(* Logix 5000 project; controller Planta_de_Kumis vendor 1 type 14 code 54 rev 20.11; software revision 20.00 *)

TASK Mapeo_IO (periodic, rate 10 ms, priority 6, watchdog 500 ms) : Mapeo_CadSim_Plus
TASK Rutina (periodic, rate 50 ms, priority 8, watchdog 500 ms) : MainProgram

MODULES
   Local : vendor 1 type 14 code 54 (ICP 0, rev 20.11)
END_MODULES

VAR_GLOBAL   (* controller tags *)
   Azucar : BOOL;
   Cultivo : BOOL;
   CV_TCV_201_1 : REAL;
   CV_TCV_202_1 : REAL;
   FI_01 : REAL;   // Indicador de flujo del vapor Intercambiador 1
   FI_02 : REAL;   // Indicador de flujo del agua Intercambiador 2
   FT_1 : REAL;
   HV2 : REAL;   // Valvula de desfogue
   HV3 : REAL;   // Valvula de desfogue TK2
   HV4 : REAL;   // Valvula de desfogue TK3
   HV5 : REAL;   // Valvula de desfogue TK4
   HV6 : REAL;   // Valvula de desfogue TK5
   HV7 : REAL;   // Valvula de desfogue TK6
   HV8 : REAL;   // Valvula de desfogue TK7
   HV9 : REAL;   // Valvula de desfogue TK8
   JY_01 : BOOL;   // Motor de mezclado M1
   JY_02 : BOOL;   // Motor de mezclado cultivo
   KP_A : REAL;   // KP de letapa de aumento de temperatura
   KP_D : REAL;   // KP de etapa de disminucion de temperatura
   Leve_TK1 : REAL;   // Sensor de nivel TK1
   Level_TK10 : REAL;   // Sensor de nivel TK10 Intercambiador 2
   Level_TK2 : REAL;   // Sensor de nivel TK2
   Level_TK3 : REAL;   // Sensor de nivel TK·
   Level_TK4 : REAL;   // Sensor de nivel TK4
   Level_TK5 : REAL;   // Sensor de nivel TK5
   Level_TK6 : REAL;   // Sensor de nivel TK6
   Level_TK7 : REAL;   // Sensor de nivel TK7
   Level_TK8 : REAL;   // Sensor de nivel TK8
   Level_TK9 : REAL;   // Sensor de nivel TK9 Intercambiador 1
   LSH_101_1 : BOOL;   // Sensor de nivel alto TK1
   LSH_102_1 : BOOL;   // Sensor de nivel alto TK2
   LSH_103_1 : BOOL;   // Sensor de nivel alto TK3
   LSH_104_1 : BOOL;   // Sensor de nivel alto TK4
   LSH_105_1 : BOOL;   // Sensor de nivel alto TK5
   LSH_106_1 : BOOL;   // Sensor de nivel alto TK6
   LSH_107_1 : BOOL;   // Sensor de nivel alto TK7
   LSH_108_1 : BOOL;   // Sensor de nivel alto TK8
   LSL_101_1 : BOOL := 1;   // Sensor de nivel bajo TK1
   LSL_102_1 : BOOL := 1;   // Sensor de nivel bajo TK2
   LSL_103_1 : BOOL := 1;   // Sensor de nivel bajo TK3
   LSL_104_1 : BOOL := 1;   // Sensor de nivel bajo TK4
   LSL_105_1 : BOOL := 1;   // Sensor de nivel bajo TK5
   LSL_106_1 : BOOL := 1;   // Sensor de nivel bajo TK6
   LSL_107_1 : BOOL := 1;   // Sensor de nivel baj TK7
   LSL_108_1 : BOOL := 1;   // Sensor de nivel bajo TK8
   PI_01 : REAL;   // Indicador de presion del vapor Intercambiador 1
   PI_02 : REAL;   // Indicador de presion del agua Intercambiador 2
   PP1 : BOOL;   // Motobomba 1
   PP2 : BOOL;   // Motobomba 2
   PP3 : BOOL;   // Motobomba 3
   PP4 : BOOL;   // Motobomba 4
   PP5 : BOOL;   // Motobomba 5
   Reset : BOOL;
   SP_A : REAL;   // SETPOINT de letapa de aumento de temperatura
   SP_D : REAL;   // SETPOINT de etapa de disminucion de temperatura
   Start : BOOL;   // Boton de Inicio
   SV_101_1 : REAL;   // Valvula de salida TK1
   SV_102_1 : REAL;   // Valvula de salida TK2
   SV_103_1 : REAL;   // Valvula de salida TK3
   SV_104_1 : REAL;   // Valvula de salida
   SV_105_1 : REAL;   // Valvula de entrada TK5
   SV_106_1 : REAL;   // Valvula de entrada TK6
   SV_107_1 : REAL;   // Valvula de entrada TK7
   SV_108_1 : REAL;   // Valvula de entrada TK8
   SV_201_1 : REAL;   // Valvula de salida 1 Intercambiador
   SV_201_2 : REAL;   // Valvula de reflujo Intercambiador 1
   SV_202_1 : REAL;   // Valvula de salida 1 Intercambiador 2
   SV_202_2 : REAL;   // Valvula de reflujo
   T_Agua : DINT := 4;   // Temperatura de entrada del Agua Fria
   T_Int : DINT := 18;   // Temperatura de entrada de la leche
   TCV_101_1 : REAL;   // Valvula de entrada de Leche Variable manipulada
   TCV_201_1 : REAL;
   TCV_202_1 : REAL;   // Valvula de entrada de agua Variable manipulada Intercambiador 2
   TD_A : REAL;   // TD de letapa de aumento de temperatura
   TD_D : REAL;   // TD de etapa de disminucion de temperatura
   TI_01 : REAL;   // Indicador de temperatura TK1
   TI_02 : REAL;   // Indicador de temperatura TK2
   TI_03 : REAL;   // Indicador de temperatura del vapor Intercambiador 1
   TI_05 : REAL;   // Indicador de temperatura TK3
   TI_06 : REAL;   // Indicador de temperatura del agua
   TI_A : REAL;   // TI de letapa de aumento de temperatura
   TI_D : REAL;   // TI de etapa de disminucion de temperatura
   TITE_201_1 : REAL;   // Sensor de temperatura de producto intermedio Variable Controlada Intercambiador 1
   TITE_202_1 : REAL;   // Sensor de temperatura de producto intermedio Variable controlada Intercambiador 2
   TITE_Prueba : REAL;
   TITE_Prueba_2 : REAL;
END_VAR

PROGRAM MainProgram   (* main routine MainRoutine *)
VAR
   a1_A : REAL;   // parametro del modelo del proceso discreto
   a1_D : REAL;   // Parametro del modelo del proceso discreto etapa de disminucion de temperatura
   aF1_A : REAL;   // Parametro delnumerador del filtro 1
   aF2_A : REAL;   // Parametro del filtro1
   b0_A : REAL;   // parametro del modelo del proceso discreto
   b0_D : REAL;   // Parametro del modelo del proceso discreto etapa de disminucion de temperatura
   b1_A : REAL;   // Parametros del modelo discreto del proceso
   b1_D : REAL;   // Parametro del modelo del proceso discreto etapa de disminucion de temperatura
   bF0_A : REAL;   // Parametro del filtro 1
   bF1_A : REAL;   // Parametro del filtro 1
   bF2_A : REAL;   // Parametro del filtro 1
   BIT_ACT : BOOL;   // BIT DE ACTIVACION ETAPA 0
   BIT_ACT2 : BOOL;   // BIT DE ACTIVACION ETAPA 0 Disminucion de temperatura
   BIT_MEZC_AZUCAR : BOOL;   // Indicador de mezclado de azucar
   BIT_MEZC_CULTIVO : BOOL;   // Bit indicador mezclado de cultivo
   BIT_PRUEBA : BOOL;
   BIT_PRUEBA_2 : BOOL;
   C1 : COUNTER := (PRE := 5);
   da : DINT;   // Retardo discreo etapa de aumento de temperatura
   dd : DINT;   // Retardo discreo etapa de disminucion de temperatura
   E0_A : REAL;   // Error actual en etapa de aumento de temperatura
   E0_D : REAL;   // Error actual en etapa de disminucion de temperatura
   E1_A : REAL;   // Error 1 instante pasado etapa de aumento de temperatura
   E1_D : REAL;   // Error 1 instante pasado etapa de disminucion de temperatura
   E2_A : REAL;   // Error 2 instantes pasados etapa de aumento de temperatura
   E2_D : REAL;   // Error 2 instantes pasados etapa de disminucion de temperatura
   Ep1_A : REAL;   // Error de prediccion 1 instante antes
   Ep2_A : REAL;   // Error de prediccion 2 instantes antes
   Ep_A : REAL;   // Error de prediccion etapa de aumento de temperatura
   Ep_D : REAL;   // Error de prediccion etapa de disminucion de temperatura
   ETAPA0_A : BOOL;   // Etapa 0 en etapa de aumento de temperatura
   ETAPA0_D : BOOL;   // Etapa 0 en etapa de disminucion de temperatura
   ETAPA10_A : BOOL;   // Etapa 10 de etapa de aumento de temperatura
   ETAPA10_D : BOOL;   // Etapa 10 en etapa de disminucion de temperatura
   ETAPA11_A : BOOL;   // Etapa 11 de etapa de aumento de temperatura
   ETAPA11_D : BOOL;   // Etapa 11 en etapa de disminucion de temperatura
   ETAPA12_A : BOOL;   // Etapa 12 de etapa de aumento de temperatura
   ETAPA12_D : BOOL;   // Etapa 12 en etapa de disminucion de temperatura
   ETAPA13_A : BOOL;   // Etapa 13 de etapa de aumento de temperatura
   ETAPA13_D : BOOL;   // Etapa 13 en etapa de disminucion de temperatura
   ETAPA14_A : BOOL;   // Etapa 14 en etapa de aumento de temperatura
   ETAPA14_D : BOOL;   // Etapa 14 en etapa de disminucion de temperatura
   ETAPA1_A : BOOL;   // Etapa 1 en etapa de aumento de temperatura
   ETAPA1_D : BOOL;   // Etapa 1 en etapa de disminucion de temperatura
   ETAPA2_A : BOOL;   // Etapa 2 en etapa de aumento de temperaura
   ETAPA2_D : BOOL;   // Etapa 2 en etapa de disminucion de temperatura
   ETAPA3_A : BOOL;   // Etapa 3 en etapa de aumento de temperatura
   ETAPA3_D : BOOL;   // Etapa 3 en etapa de disminucion de temperatura
   ETAPA4_A : BOOL;   // Etapa 4 en etapa de aumento de temperatura
   ETAPA4_D : BOOL;   // Etapa 4 en etapa de disminucion de temperatura
   ETAPA5_A : BOOL;   // Etapa 5 de etapa de aumento de temperatura
   ETAPA5_D : BOOL;   // Etapa 5 en etapa de disminucion de temperatura
   ETAPA6_A : BOOL;   // Etapa 6 de etapa de aumento de temperatura
   ETAPA6_D : BOOL;   // Etapa 6 en etapa de disminucion de temperatura
   ETAPA7_A : BOOL;   // Etapa 7 en etapa de aumento de temperatura
   ETAPA7_D : BOOL;   // Etapa 7 en etapa de disminucion de temperatura
   ETAPA8_A : BOOL;   // Etapa 8 en etapa de aumento de temperatura
   ETAPA8_D : BOOL;   // Etapa 8 en etapa de disminucion de temperatura
   ETAPA9_A : BOOL;   // Etapa 9 de etapa de aumento de temperatura
   ETAPA9_D : BOOL;   // Etapa 9 en etapa de disminucion de temperatura
   I_A : DINT;   // Indice etapa de aumento de temperatura
   I_D : DINT;   // Indice etapa de disminucion de temperatura
   KTA : DINT;   // Tiempo discreto actual ultima posicion del vector U etapa de aumento
   KTD : DINT;   // Tiempo discreto actual ultima posicion del vector U etapa de disminucion de temperatura
   Latch_Azcuar_On : BOOL;
   Latch_LSH_TK1 : BOOL;
   Latch_LSH_TK2 : BOOL;
   Latch_LSH_TK3 : BOOL;
   Latch_LSH_TK4 : BOOL;
   Latch_LSH_TK5 : BOOL;
   Latch_LSH_TK6 : BOOL;
   Latch_LSH_TK7 : BOOL;
   Latch_LSH_TK8 : BOOL;
   Latch_OSR_2 : BOOL;
   Latch_OSR_4 : BOOL;
   Latch_OSR_6 : BOOL;
   Latch_OSR_8 : BOOL;
   Latch_PID2 : BOOL;
   Latch_SR1 : BOOL;
   Latch_SR2 : BOOL;
   Latch_Timer_Mezclado_DN : BOOL;
   Next_Batch : BOOL;
   OSR_1 : BOOL;
   OSR_2 : BOOL;
   OSR_3 : BOOL;
   OSR_4 : BOOL;
   OSR_5 : BOOL;
   OSR_6 : BOOL;
   OSR_7 : BOOL;
   OSR_8 : BOOL;
   OSRI_1 : FBD_ONESHOT;   // PULSO
   OSRI_2 : FBD_ONESHOT;   // Pulso
   PID_Exchanger_1 : PID := (CTL := 142607488, DOE := 1, PE := 1, DVNA := 1, PVHA := 1, SP := 60.0, MAXS := 100.0, MINS := 18.0, MAXO := 100.0, UPD := 1.0, MAXI := 100.0, MINI := 18.0, MAXCV := 100.0, DATA[0] := 45.327106, DATA[1] := -1256.7006, DATA[2] := 117.815674, DATA[3] := -57.815674, DATA[4] := 60.0, DATA[5] := 0.6666667, DATA[6] := 1.0, DATA[7] := 0.8, DATA[8] := 0.51, DATA[9] := 0.018, DATA[11] := 0.51, DATA[12] := 0.018, DATA[15] := 1.5, DATA[16] := 0.024420025);   // PID para el intercambiado de calor con vapor
   PID_Exchanger_2 : PID := (CTL := 176165504, DOE := 1, CA := 1, PE := 1, OLH := 1, DVPA := 1, PVHA := 1, SP := 40.0, MAXS := 100.0, SO := 100.0, MAXO := 100.0, UPD := 1.0, ERR := 39.804905, MAXI := 100.0, MAXCV := 100.0, DATA[0] := 65.07602, DATA[1] := -0.31215367, DATA[2] := 0.19509344, DATA[3] := 39.804905, DATA[4] := 40.0, DATA[5] := 0.1, DATA[6] := 1.0, DATA[7] := 33.989998, DATA[8] := 0.013, DATA[9] := 71.98, DATA[10] := 17.99, DATA[11] := 0.013, DATA[12] := 71.98, DATA[13] := 17.99, DATA[15] := 10.0, DATA[16] := 0.024420025);   // PID para el intercambiador de disminucion de temperatura
   q0_A : REAL;   // Parametro del controlador PID digital
   q0_D : REAL;   // Parametro del controlador PID digital etapa de disminucion de temperatura
   q1_A : REAL;   // Parametros del controlador PID digital
   q1_D : REAL;   // Parametro del controlador PID digital etapa de disminucion de temperatura
   q2_A : REAL;   // Parametros del controlador PID digital
   q2_D : REAL;   // Parametro del controlador PID digital etapa de disminucion de temperatura
   Salida_Prueba_1 : BOOL;
   TIMER_AT : FBD_TIMER;   // Timer de espera para mover datos en el vector de esfuerzo de control etapa de aumento de temperatura
   Timer_Azucar : TIMER := (PRE := 1000);
   Timer_Cultivo : TIMER := (PRE := 1000);
   Timer_Disminucion_T : TIMER := (PRE := 1000);
   TIMER_DT : FBD_TIMER;   // Timer de espera para mover datos en el vector de esfuerzo de control etapa de disminucion de temperatura
   timer_Elevado_T : TIMER := (PRE := 1000);
   Timer_Inoculado : TIMER := (PRE := 6000);
   Timer_Latch_PID2 : TIMER := (PRE := 42000);   // Timer para activacion del PID 2
   Timer_Mezclado : TIMER := (PRE := 1000);
   Timer_Recepcion : TIMER := (PRE := 1000);
   Timer_TK5 : TIMER := (PRE := 5000);
   Timer_TK6 : TIMER := (PRE := 5000);
   Timer_TK7 : TIMER := (PRE := 5000);
   Timer_TK8 : TIMER := (PRE := 5000);
   Tm_A : REAL;   // Tiempo de muestreo etapa aumento de temperatura
   Tm_D : REAL;   // Tiempo de muestreo etapa disminucion de temperatura
   VEC_U_A : REAL[24];   // VECTOR DE ESFUERZO DE CONTROL de etapa de aumento de temperatura
   VEC_U_D : REAL[24];   // VECTOR DE ESFUERZO DE CONTROL de etapa de disminucion de temperatura
   yF1_A : REAL;   // salida del filtro 1 instante antes
   yF2_A : REAL;   // salida del filtro 1 endos instantes antes
   yF_A : REAL;   // Salida del filtro 1
   Yn1_A : REAL;   // Salida del modelo nominal (Con retardo) 1 instante antes etapa de aumento de temparatura
   Yn1_D : REAL;   // Salida del modelo nominal (Con retardo) 1 instante antes etapa de disminucion de temperatura
   Yn_A : REAL;   // Salida del modelo nominal (Con retardo) etapa de aumento de temperatura
   Yn_D : REAL;   // Salida del modelo nominal (Con retardo) etapa de disminucion de temperatura
   Yp_A : REAL;   // Salida predicha etapa de aumento de temperatura
   Yp_D : REAL;   // Salida predicha etapa de disminucion de temperatura
   Yt1_A : REAL;   // Salida del modelo nominal rapido (Sin retardo) 1 instante antes etapa de aumento de temperatura
   Yt1_D : REAL;   // Salida del modelo nominal rapido (Sin retardo) 1 instante antes etapa de disminucion de temperatura
   Yt_A : REAL;   // Salida del modelo nominal rapido (Sin retardo) etapa de aumento de temperatura
   Yt_D : REAL;   // Salida del modelo nominal rapido (Sin retardo) etapa de disminucion de temperatura
END_VAR

ROUTINE MainRoutine   (* ladder *)
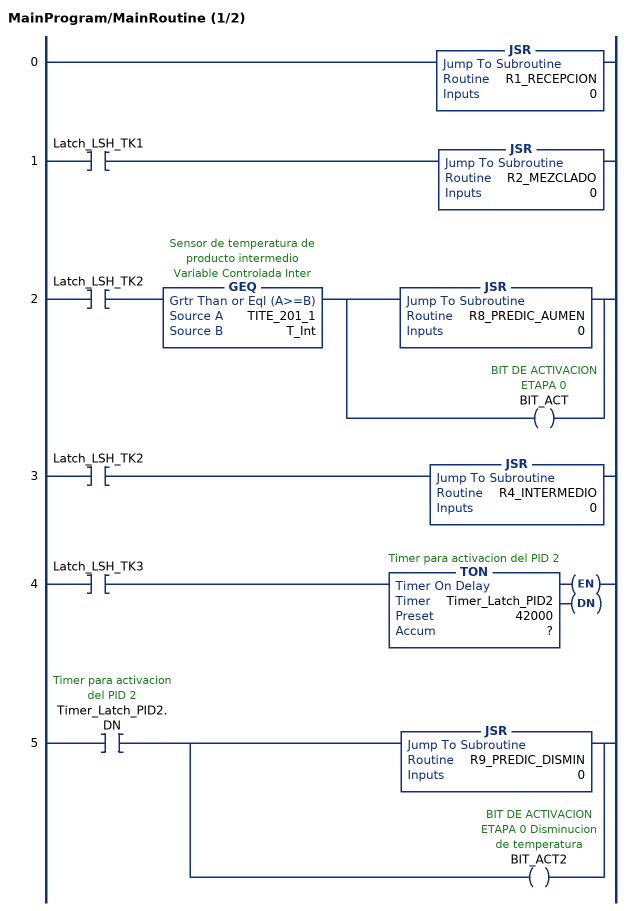
   0: JSR(R1_RECEPCION,0);
   1: XIC(Latch_LSH_TK1)JSR(R2_MEZCLADO,0);
   2: XIC(Latch_LSH_TK2)GEQ(TITE_201_1,T_Int)[JSR(R8_PREDIC_AUMEN,0) ,OTE(BIT_ACT) ];
   3: XIC(Latch_LSH_TK2)JSR(R4_INTERMEDIO,0);
   4: XIC(Latch_LSH_TK3)TON(Timer_Latch_PID2,?,?);
   5: XIC(Timer_Latch_PID2.DN)[JSR(R9_PREDIC_DISMIN,0) ,OTE(BIT_ACT2) ];
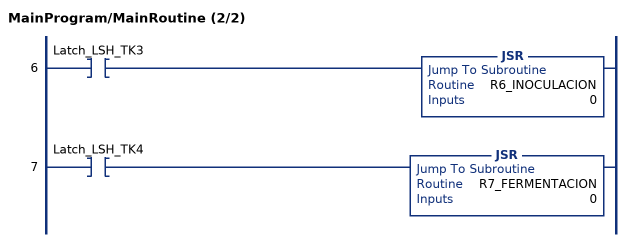
   6: XIC(Latch_LSH_TK3)JSR(R6_INOCULACION,0);
   7: XIC(Latch_LSH_TK4)JSR(R7_FERMENTACION,0);
END_ROUTINE

ROUTINE R11_BLOQUE_PREDICTOR1   (* structured text *)
   // BLOQUE PREDICTOR DE SMITH - ETAPA DE AUMENTO DE TEMPERATURA
   
   OSRI_1.InputBit :=  BIT_ACT;
   OSRI(OSRI_1);
   IF (OSRI_1.OutputBit) THEN
   ETAPA0_A :=1;
   END_IF;
   
   IF ETAPA0_A AND NOT ETAPA2_A THEN
   ETAPA0_A := 0;
   ETAPA1_A := 1;
   END_IF;
   
   IF ETAPA1_A THEN
   // INICIALIZACION DE VARIABLES
   KTA:=23;   // Ultima posicion del vector de esfuerzo de control
   da := 22;  // Retardo discreto
   I_A := 1;  // Indice
   
   b0_A := 0;    // b0, b1 y a1 parametros del modelo del proceso
   b1_A := 0.098;
   a1_A := -0.8948;
   //TCV_201_1 := 5;
   E0_A := 0;  // Error actual
   Ep_A := 0; // Error de prediccion
   
   Yp_A := 0; //  Salida predicha
   Yn_A := TITE_201_1; // Salida del modelo nominal (Con retardo)
   Yn1_A := TITE_201_1; // Salida del modelo nominal (Con retardo) 1 instante antes
   Yt_A := TITE_201_1;  // Salida del modelo nominal rapido (Sin retardo)
   Yt1_A := TITE_201_1;  // Salida del modelo nominal rapido (Sin retardo) 1 instante antes
   (*
   // Inicializacion del vector de esfuerzo de control
   	FOR I_A:=0 TO 23 DO
   	VEC_U_A[I_A] := 5;
   	END_FOR;
   *)
   END_IF;
   
   IF (ETAPA1_A AND NOT ETAPA3_A) OR (ETAPA10_A AND TIMER_AT.DN) THEN
   ETAPA1_A := 0;
   ETAPA2_A := 1;
   ETAPA10_A := 0;
   I_A :=1;
   TIMER_AT.Reset := 1;
   TIMER_AT.TimerEnable := 0;
   END_IF;
   
   IF ETAPA2_A THEN
   // SALIDA DEL MODELO NOMINAL CON RETARDO
   Yn_A := (b0_A * VEC_U_A[KTA - da]) + (b1_A * VEC_U_A[KTA - 1 - da]) -  (a1_A * Yn1_A);
   END_IF;
   
   IF ETAPA2_A AND NOT ETAPA4_A THEN
   ETAPA2_A := 0;
   ETAPA3_A := 1;
   END_IF;
   
   IF ETAPA3_A THEN
   // ERROR DE PREDICCION : DIFERENCIA ENTRE EL PROCESO REAL Y NOMINAL
   Ep_A := TITE_201_1 - Yn_A;
   END_IF;
   
   IF ETAPA3_A AND NOT ETAPA5_A THEN
   ETAPA3_A := 0;
   ETAPA4_A := 1;
   END_IF;
   
   IF ETAPA4_A THEN
   // MODELO NOMINAL RAPIDO (SIN RETARDO)
   Yt_A := (b0_A * VEC_U_A[KTA]) + (b1_A * VEC_U_A[KTA - 1])  -  (a1_A * Yt1_A);
   END_IF;
   
   IF ETAPA4_A AND NOT ETAPA6_A THEN
   ETAPA4_A := 0;
   ETAPA5_A := 1;
   END_IF;
   
   IF ETAPA5_A THEN
   // SUMA DEL ERROR DE PREDICCION Y LA SALIDA DEL MODELO NOMINAL RAPIDO (SIN RETARDO)
   Yp_A := Yt_A + Ep_A;
   END_IF;
   
   IF ETAPA5_A AND NOT ETAPA7_A THEN
   ETAPA5_A := 0;
   ETAPA6_A := 1;
   END_IF;
   
   IF ETAPA6_A THEN
   // CALCULO DEL ERROR: ERROR = SETPOINT - Yp
   PID_Exchanger_1.ERR := PID_Exchanger_1.SP - Yp_A;
   END_IF;
   
   IF ETAPA6_A AND NOT ETAPA8_A THEN
   ETAPA6_A := 0;
   ETAPA7_A := 1;
   END_IF;
   
   IF ETAPA7_A THEN
   VEC_U_A[KTA] := TCV_201_1;
   END_IF;
   
   IF ETAPA7_A AND NOT ETAPA9_A THEN
   ETAPA7_A := 0;
   ETAPA8_A := 1;
   END_IF;
   
   IF ETAPA8_A THEN			// Desplazamiento de valores en el vector de la ley de control
   	FOR I_A:=1 TO KTA DO
   		VEC_U_A[I_A - 1] := VEC_U_A[I_A];
   	END_FOR;
   END_IF;
   
   IF ETAPA8_A AND NOT ETAPA10_A THEN
   ETAPA8_A := 0;
   ETAPA9_A := 1;
   END_IF;
   
   IF ETAPA9_A THEN
   Yn1_A := Yn_A;
   Yt1_A := Yt_A;
   END_IF;
   
   IF ETAPA9_A AND NOT ETAPA2_A THEN
   ETAPA9_A := 0;
   ETAPA10_A := 1;
   END_IF;
   
   IF ETAPA10_A THEN
   TONR(TIMER_AT);
   TIMER_AT.PRE := 1000;
   TIMER_AT.Reset := 0;
   TIMER_AT.TimerEnable := 1;
   END_IF;
END_ROUTINE

ROUTINE R12_BLOQUE_PREDICTOR2   (* structured text *)
   // PREDICTOR DE SMITH - ETAPA DE DISMINUCION DE TEMPERATURA
   
   OSRI_2.InputBit :=  BIT_ACT2;
   OSRI(OSRI_2);
   IF (OSRI_2.OutputBit) THEN
   ETAPA0_D :=1;
   END_IF;
   
   IF ETAPA0_D AND NOT ETAPA2_D THEN
   ETAPA1_D := 1;
   ETAPA0_D := 0;
   END_IF;
   
   IF ETAPA1_D THEN
   // INICIALIZACIONDE VARIABLES
   KTD:=23;    // Ultima pocicion del vector de esfuerzo de control
   dd := 21;   // Retardo discreto
   I_D := 1;  // Indice
   
   b0_D :=0;		// b0, b1 y a1 parametros del modelo del proceso
   b1_D := 0.047;
   a1_D := -0.9355;
   
   Ep_D := 0; // Error de prediccion
   
   Yp_D := 0; //  Salida predicha
   Yn_D := TITE_202_1; // Salida del modelo nominal (Con retardo)
   Yn1_D := TITE_202_1; // Salida del modelo nominal (Con retardo) 1 instante antes
   Yt_D := TITE_202_1;  // Salida del modelo nominal rapido (Sin retardo)
   Yt1_D := TITE_202_1;  // Salida del modelo nominal rapido (Sin retardo) 1 instante antes
   
   // Inicializacion del vector de esfuerzo de control
   	FOR I_D:=0 TO 23 DO
   	VEC_U_D[I_D] := 0;
   	END_FOR;
   END_IF;
   
   IF (ETAPA1_D AND NOT ETAPA3_D) OR ETAPA9_D THEN
   ETAPA1_D := 0;
   ETAPA2_D := 1;
   ETAPA9_D := 0;
   I_D :=1;
   END_IF;
   
   IF ETAPA2_D THEN
   // SALIDA DEL MODELO NOMINAL CON RETARDO
   Yn_D := (b0_D * VEC_U_D[KTD - dd]) + (b1_D * VEC_U_D[KTD - 1 - dd]) -  (a1_D * Yn1_D);  // 	Calcula la salida del modelo nominal (con retardo)
   END_IF;
   
   IF ETAPA2_D AND NOT ETAPA4_D THEN
   ETAPA2_D := 0;
   ETAPA3_D := 1;
   END_IF;
   
   IF ETAPA3_D THEN
   // ERROR DE PREDICCION : DIFERENCIA ENTRE EL PROCESO REAL Y NOMINAL
   Ep_D := TITE_202_1 - Yn_D;  // Calculo del error de prediccion - Diferencia entre el proceso real y el proceso nominal
   END_IF;
   
   IF ETAPA3_D AND NOT ETAPA5_D THEN
   ETAPA3_D := 0;
   ETAPA4_D := 1;
   END_IF;
   
   IF ETAPA4_D THEN
   // MODELO NOMINAL RAPIDO (SIN RETARDO)
   Yt_D := (b0_D * VEC_U_D[KTD]) + (b1_D * VEC_U_D[KTD - 1])  -  (a1_D * Yt1_D);  // Calculo de la salida del modelo nominal rapido (sin retardo)
   END_IF;
   
   IF ETAPA4_D AND NOT ETAPA6_D THEN
   ETAPA4_D := 0;
   ETAPA5_D := 1;
   END_IF;
   
   IF ETAPA5_D THEN
   // SUMA DEL ERROR DE PREDICCION Y LA SALIDA DEL MODELO NOMINAL RAPIDO (SIN RETARDO)
   Yp_D := Yt_D + Ep_D;  // Suma emtre el error de prediccion y la salida del modelo nominal rapido (sin retardo)
   END_IF;
   
   IF ETAPA5_D AND NOT ETAPA7_D THEN
   ETAPA5_D := 0;
   ETAPA6_D := 1;
   END_IF;
   
   IF ETAPA6_D THEN
   PID_Exchanger_2.ERR := Yp_D - PID_Exchanger_2.SP;
   END_IF;
   
   IF ETAPA6_D AND NOT ETAPA8_D THEN
   ETAPA6_D := 0;
   ETAPA7_D := 1;
   END_IF;
   
   IF ETAPA7_D THEN
   VEC_U_D[KTD] := TCV_202_1;
   END_IF;
   
   IF ETAPA7_D AND NOT ETAPA9_D THEN
   ETAPA7_D := 0;
   ETAPA8_D := 1;
   END_IF;
   
   IF ETAPA8_D THEN			// Desplazamiento de valores en el vector de la ley de control
   	FOR I_D:=1 TO KTD DO
   		VEC_U_D[I_D - 1] := VEC_U_D[I_D];
   	END_FOR;
   END_IF;
   
   IF ETAPA8_D AND NOT ETAPA2_D THEN
   ETAPA8_D := 0;
   ETAPA9_D := 1;
   END_IF;
   
   IF ETAPA9_D THEN
   Yn1_D := Yn_D;
   Yt1_D := Yt_D;
   END_IF;
   
END_ROUTINE

ROUTINE R1_RECEPCION   (* ladder *)
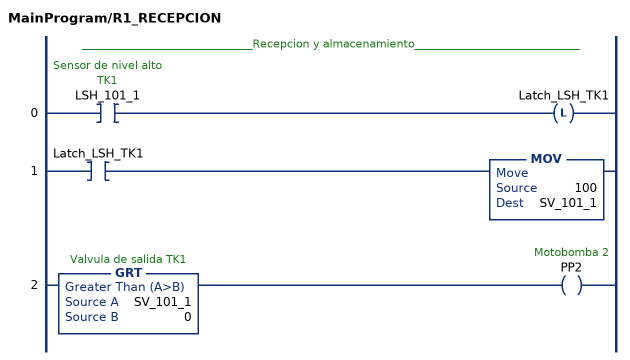
   // _______________________________Recepcion y almacenamiento______________________________
   0: XIC(LSH_101_1)OTL(Latch_LSH_TK1);
   1: XIC(Latch_LSH_TK1)MOV(100,SV_101_1);
   2: GRT(SV_101_1,0)OTE(PP2);
END_ROUTINE

ROUTINE R2_MEZCLADO   (* ladder *)
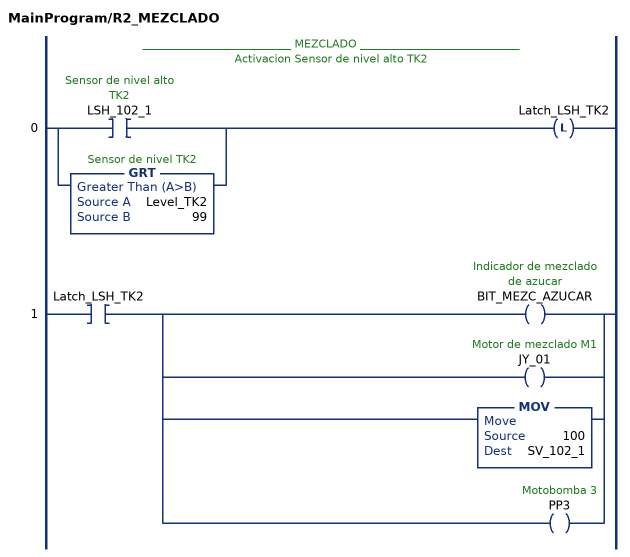
   // ___________________________ MEZCLADO _____________________________
   // Activacion Sensor de nivel alto TK2
   0: [XIC(LSH_102_1) ,GRT(Level_TK2,99) ]OTL(Latch_LSH_TK2);
   1: XIC(Latch_LSH_TK2)[OTE(BIT_MEZC_AZUCAR) ,[OTE(JY_01) ,[MOV(100,SV_102_1) ,OTE(PP3) ] ] ];
END_ROUTINE

ROUTINE R3_AUMENTO_TEMP   (* ladder *)
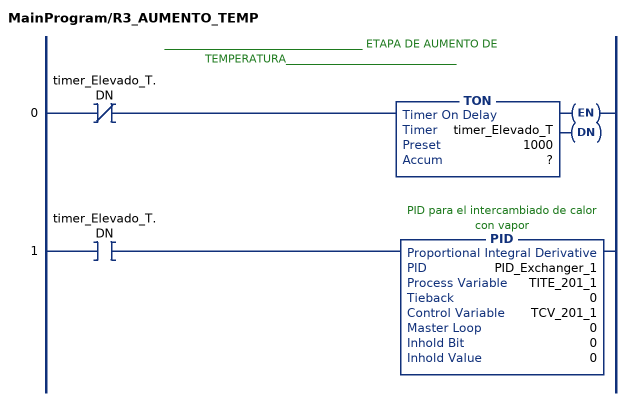
   // ____________________________________ ETAPA DE AUMENTO DE TEMPERATURA_______________________________
   0: XIO(timer_Elevado_T.DN)TON(timer_Elevado_T,?,?);
   1: XIC(timer_Elevado_T.DN)PID(PID_Exchanger_1,TITE_201_1,0,TCV_201_1,0,0,0);
END_ROUTINE

ROUTINE R4_INTERMEDIO   (* ladder *)
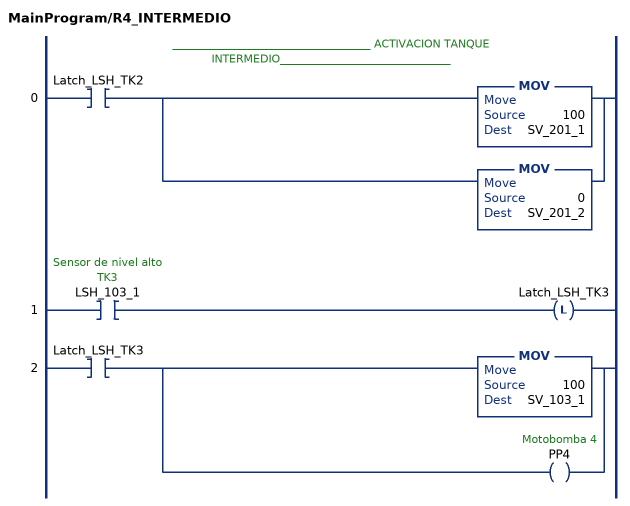
   // ____________________________________ ACTIVACION TANQUE INTERMEDIO_______________________________
   0: XIC(Latch_LSH_TK2)[MOV(100,SV_201_1) ,MOV(0,SV_201_2) ];
   1: XIC(LSH_103_1)OTL(Latch_LSH_TK3);
   2: XIC(Latch_LSH_TK3)[MOV(100,SV_103_1) ,OTE(PP4) ];
END_ROUTINE

ROUTINE R5_DISMINUCION_TEMP   (* ladder *)
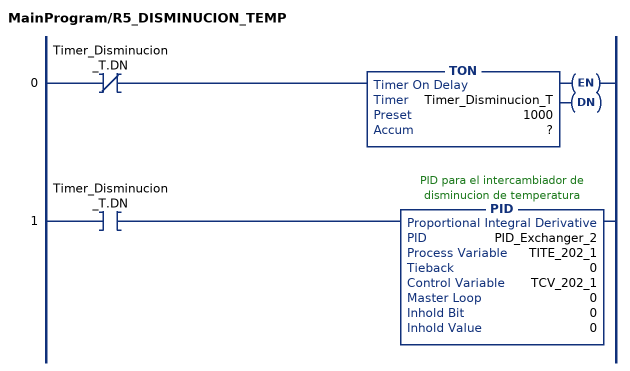
   0: XIO(Timer_Disminucion_T.DN)TON(Timer_Disminucion_T,?,?);
   1: XIC(Timer_Disminucion_T.DN)PID(PID_Exchanger_2,TITE_202_1,0,TCV_202_1,0,0,0);
END_ROUTINE

ROUTINE R6_INOCULACION   (* ladder *)
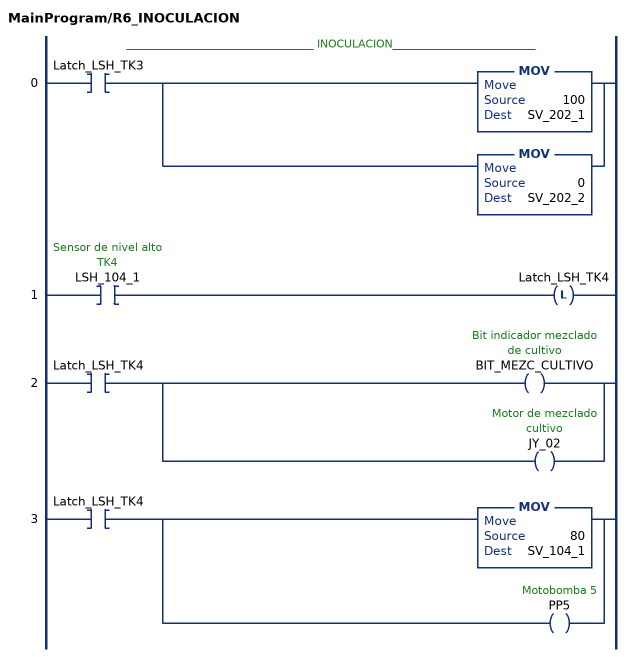
   // __________________________________ INOCULACION__________________________
   0: XIC(Latch_LSH_TK3)[MOV(100,SV_202_1) ,MOV(0,SV_202_2) ];
   1: XIC(LSH_104_1)OTL(Latch_LSH_TK4);
   2: XIC(Latch_LSH_TK4)[OTE(BIT_MEZC_CULTIVO) ,OTE(JY_02) ];
   3: XIC(Latch_LSH_TK4)[MOV(80,SV_104_1) ,OTE(PP5) ];
END_ROUTINE

ROUTINE R7_FERMENTACION   (* ladder *)
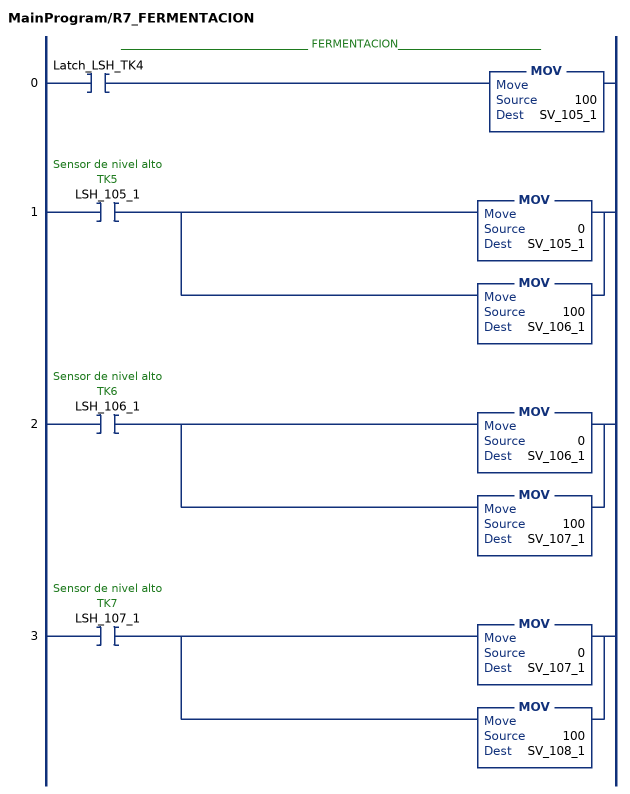
   // __________________________________ FERMENTACION__________________________
   0: XIC(Latch_LSH_TK4)MOV(100,SV_105_1);
   1: XIC(LSH_105_1)[MOV(0,SV_105_1) ,MOV(100,SV_106_1) ];
   2: XIC(LSH_106_1)[MOV(0,SV_106_1) ,MOV(100,SV_107_1) ];
   3: XIC(LSH_107_1)[MOV(0,SV_107_1) ,MOV(100,SV_108_1) ];
END_ROUTINE

ROUTINE R8_PREDIC_AUMEN   (* structured text *)
   // PREDICTOR DE SMITH - ETAPA DE AUMENTO DE TEMPERATURA
   // BIT DE ACTIVACION
   OSRI_1.InputBit :=  BIT_ACT;
   OSRI(OSRI_1);
   IF (OSRI_1.OutputBit) THEN
   ETAPA0_A :=1;
   END_IF;
   
   IF ETAPA0_A AND NOT ETAPA2_A THEN
   ETAPA1_A := 1;
   ETAPA0_A := 0;
   END_IF;
   
   IF ETAPA1_A THEN
   // INICIALIZACION DE VARIABLES
   KTA:=23;   // Ultima posicion del vector de esfuerzo de control
   da := 22;  // Retardo discreto
   I_A := 1;  // Indice
   Tm_A := 1;  // Tiempo de muestreo
   q0_A := 0;  // q0, q1 y q2 Parametros del controlador PID digital
   q1_A := 0;
   q2_A := 0;
   
   b0_A := 0;    // b0, b1 y a1 parametros del modelo del proceso
   b1_A := 0.098;
   a1_A := -0.8948;
   
   E0_A := 0;  // Error actual
   E1_A := 0;  // Error 1 instante pasado
   E2_A := 0;  // Error 2 instantes pasado
   
   Ep_A := 0; // Error de prediccion
   
   Yp_A := 0; //  Salida predicha
   Yn_A := TITE_201_1; // Salida del modelo nominal (Con retardo)
   Yn1_A := TITE_201_1; // Salida del modelo nominal (Con retardo) 1 instante antes
   Yt_A := TITE_201_1;  // Salida del modelo nominal rapido (Sin retardo)
   Yt1_A := TITE_201_1;  // Salida del modelo nominal rapido (Sin retardo) 1 instante antes
   
   // Inicializacion del vector de esfuerzo de control
   	FOR I_A:=0 TO 23 DO
   	VEC_U_A[I_A] := 0;
   	END_FOR;
   // Calculo de parametros q0, q1, q2 del controlador digital
   q0_A := KP_A * (1 +  Tm_A/(2*TI_A)  +   TD_A/Tm_A);
   q1_A := -KP_A * (1 -  Tm_A/(2*TI_A)  +   (2*TD_A)/Tm_A);
   q2_A := (KP_A * TD_A)/Tm_A;
   END_IF;
   
   IF (ETAPA1_A AND NOT ETAPA3_A) OR (ETAPA14_A AND TIMER_AT.DN) THEN
   ETAPA1_A := 0;
   ETAPA2_A := 1;
   ETAPA14_A := 0;
   TIMER_AT.Reset := 1;
   TIMER_AT.TimerEnable := 0;
   I_A :=1;
   END_IF;
   
   IF ETAPA2_A THEN
   Yn_A := (b0_A * VEC_U_A[KTA - da]) + (b1_A * VEC_U_A[KTA - 1 - da]) -  (a1_A * Yn1_A);  // 	Calcula la salida del modelo nominal (con retardo)
   END_IF;
   
   IF ETAPA2_A AND NOT ETAPA4_A THEN
   ETAPA2_A := 0;
   ETAPA3_A := 1;
   END_IF;
   
   IF ETAPA3_A THEN
   Ep_A := TITE_201_1 - Yn_A;  // Calculo del error de prediccion : Diferencia entre el proceso real y el proceso nominal
   END_IF;
   
   IF ETAPA3_A AND NOT ETAPA5_A THEN
   ETAPA3_A := 0;
   ETAPA4_A := 1;
   END_IF;
   
   IF ETAPA4_A THEN
   Yt_A := (b0_A * VEC_U_A[KTA]) + (b1_A * VEC_U_A[KTA - 1])  -  (a1_A * Yt1_A);  // Calculo de la salida del modelo nominal rapido (sin retardo)
   END_IF;
   
   IF ETAPA4_A AND NOT ETAPA6_A THEN
   ETAPA4_A := 0;
   ETAPA5_A := 1;
   END_IF;
   
   IF ETAPA5_A THEN
   Yp_A := Yt_A + Ep_A;  // Suma emtre el error de prediccion y la salida del modelo nominal rapido (sin retardo)
   END_IF;
   
   IF ETAPA5_A AND NOT ETAPA7_A THEN
   ETAPA5_A := 0;
   ETAPA6_A := 1;
   END_IF;
   
   // PID
   IF ETAPA6_A THEN
   E0_A := SP_A - Yp_A; // Calculo del error
   END_IF;
   
   IF ETAPA6_A AND NOT ETAPA8_A THEN
   ETAPA6_A := 0;
   ETAPA7_A := 1;
   END_IF;
   
   IF ETAPA7_A THEN
   VEC_U_A[KTA] := VEC_U_A[KTA - 1]  +  q0_A * E0_A  +  q1_A * E1_A  +  q2_A * E2_A;  // Ley de control
   END_IF;
   
   IF ETAPA7_A AND NOT ETAPA9_A THEN
   ETAPA7_A := 0;
   ETAPA8_A := 1;
   END_IF;
   
   IF ETAPA8_A THEN		// Saturacion de la accion del control en un valor maximo y minimo
   	IF VEC_U_A[KTA] >= 100 THEN
   		VEC_U_A[KTA] := 100;
   	END_IF;
   
   	IF VEC_U_A[KTA] <= 0 THEN
   		VEC_U_A[KTA] := 0;
   	END_IF;
   END_IF;
   
   IF ETAPA8_A AND NOT ETAPA10_A THEN
   ETAPA8_A := 0;
   ETAPA9_A := 1;
   END_IF;
   
   IF ETAPA9_A THEN
   TCV_201_1 :=  VEC_U_A[KTA];  // Envio de valor de esfuerzo de control a la valvula de vapor del intercambiador de calor 1
   END_IF;
   
   IF ETAPA9_A AND NOT ETAPA11_A THEN
   ETAPA9_A := 0;
   ETAPA10_A := 1;
   END_IF;
   
   IF ETAPA10_A THEN
   E2_A := E1_A;  // Actualizacion de errores pasados
   END_IF;
   
   IF ETAPA10_A AND NOT ETAPA12_A THEN
   ETAPA10_A := 0;
   ETAPA11_A := 1;
   END_IF;
   
   IF ETAPA11_A THEN
   E1_A := E0_A;   // Actualizacion de errores pasados
   END_IF;
   
   IF ETAPA11_A AND NOT ETAPA13_A THEN
   ETAPA11_A := 0;
   ETAPA12_A := 1;
   END_IF;
   
   IF ETAPA12_A THEN			// Desplazamiento de valores en el vector de la ley de control para actualizar valores pasados
   	FOR I_A:=1 TO KTA DO
   		VEC_U_A[I_A - 1] := VEC_U_A[I_A];
   	END_FOR;
   END_IF;
   
   IF ETAPA12_A AND NOT ETAPA14_A THEN
   ETAPA12_A := 0;
   ETAPA13_A := 1;
   END_IF;
   
   IF ETAPA13_A THEN
   Yn1_A := Yn_A;   // Actualizacion de valores pasados del modelo con retardo y el modelo rapido
   Yt1_A := Yt_A;
   END_IF;
   
   IF ETAPA13_A AND NOT ETAPA2_A THEN
   ETAPA13_A := 0;
   ETAPA14_A := 1;
   END_IF;
   
   IF ETAPA14_A THEN    //  Tiempo de espera para recibir datos
   TONR(TIMER_AT);
   TIMER_AT.PRE := 2000;
   TIMER_AT.Reset := 0;
   TIMER_AT.TimerEnable := 1;
   END_IF;
   
   
END_ROUTINE

ROUTINE R9_PREDIC_DISMIN   (* structured text *)
   // PREDICTOR DE SMITH - ETAPA DE DISMINUCION DE TEMPERATURA
   // Bit de activacion
   OSRI_2.InputBit :=  BIT_ACT2;
   OSRI(OSRI_2);
   IF (OSRI_2.OutputBit) THEN
   ETAPA0_D :=1;
   END_IF;
   
   IF ETAPA0_D AND NOT ETAPA2_D THEN
   ETAPA0_D := 0;
   ETAPA1_D := 1;
   END_IF;
   
   IF ETAPA1_D THEN
   // Actualizacion de variables
   KTD:=23;    // Ultima pocicion del vector de esfuerzo de control
   dd := 21;   // Retardo discreto
   I_D := 1;  // Indice
   Tm_D := 1;  // Tiempo de muestreo
   q0_D := 0;  // q0, q1 y q2 Parametros del controlador PID digital
   q1_D := 0;
   q2_D := 0;
   
   b0_D :=0;		// b0, b1 y a1 parametros del modelo del proceso
   b1_D := -0.047;
   a1_D := -0.9355;
   
   E0_D := 0;  // Error actual
   E1_D := 0;  // Error 1 instante pasado
   E2_D := 0;  // Error 2 instantes pasado
   
   Ep_D := 0; // Error de prediccion
   
   Yp_D := 0; //  Salida predicha
   Yn_D := TITE_202_1; // Salida del modelo nominal (Con retardo)
   Yn1_D := TITE_202_1; // Salida del modelo nominal (Con retardo) 1 instante antes
   Yt_D := TITE_202_1;  // Salida del modelo nominal rapido (Sin retardo)
   Yt1_D := TITE_202_1;  // Salida del modelo nominal rapido (Sin retardo) 1 instante antes
   
   // Inicializacion del vector de esfuerzo de control
   	FOR I_D:=0 TO 23 DO
   	VEC_U_D[I_D] := 0;
   	END_FOR;
   // Calculo de parametros q0, q1, q2 del controlador digital
   q0_D := KP_D * (1 +  Tm_D/(2*TI_D)  +   TD_D/Tm_D);
   q1_D := -KP_D * (1 -  Tm_D/(2*TI_D)  +   (2*TD_D)/Tm_D);
   q2_D := (KP_D * TD_D)/Tm_D;
   END_IF;
   
   IF (ETAPA1_D AND NOT ETAPA3_D) OR (ETAPA14_D AND TIMER_DT.DN) THEN
   ETAPA1_D := 0;
   ETAPA2_D := 1;
   ETAPA14_D := 0;
   TIMER_DT.Reset := 1;
   TIMER_DT.TimerEnable := 0;
   I_D :=1;
   END_IF;
   
   IF ETAPA2_D THEN
   Yn_D := (b0_D * VEC_U_D[KTD - dd]) + (b1_D * VEC_U_D[KTD - 1 - dd]) -  (a1_D * Yn1_D);  // 	Calcula la salida del modelo nominal (con retardo)
   END_IF;
   
   IF ETAPA2_D AND NOT ETAPA4_D THEN
   ETAPA2_D := 0;
   ETAPA3_D := 1;
   END_IF;
   
   IF ETAPA3_D THEN
   Ep_D := TITE_202_1 - Yn_D;  // Calculo del error de prediccion : Diferencia entre el proceso real y el proceso nominal
   END_IF;
   
   IF ETAPA3_D AND NOT ETAPA5_D THEN
   ETAPA3_D := 0;
   ETAPA4_D := 1;
   END_IF;
   
   IF ETAPA4_D THEN
   Yt_D := (b0_D * VEC_U_D[KTD]) + (b1_D * VEC_U_D[KTD - 1])  -  (a1_D * Yt1_D);  // Calculo de la salida del modelo nominal rapido (sin retardo)
   END_IF;
   
   IF ETAPA4_D AND NOT ETAPA6_D THEN
   ETAPA4_D := 0;
   ETAPA5_D := 1;
   END_IF;
   
   IF ETAPA5_D THEN
   Yp_D := Yt_D + Ep_D;  // Suma emtre el error de prediccion y la salida del modelo nominal rapido (sin retardo)
   END_IF;
   
   IF ETAPA5_D AND NOT ETAPA7_D THEN
   ETAPA5_D := 0;
   ETAPA6_D := 1;
   END_IF;
   
   // PID
   IF ETAPA6_D THEN
   E0_D := Yp_D - SP_D;  // Calculo del error
   END_IF;
   
   IF ETAPA6_D AND NOT ETAPA8_D THEN
   ETAPA6_D := 0;
   ETAPA7_D := 1;
   END_IF;
   
   IF ETAPA7_D THEN
   VEC_U_D[KTD] := VEC_U_D[KTD - 1]  +  q0_D * E0_D  +  q1_D * E1_D  +  q2_D * E2_D;  // Ley de control
   END_IF;
   
   IF ETAPA7_D AND NOT ETAPA9_D THEN
   ETAPA7_D := 0;
   ETAPA8_D := 1;
   END_IF;
   
   IF ETAPA8_D THEN		// Saturacion de la accion del control en un valor maximo y minimo
   	IF VEC_U_D[KTD] >= 100 THEN
   		VEC_U_D[KTD] := 100;
   	END_IF;
   
   	IF VEC_U_D[KTD] <= 0 THEN
   		VEC_U_D[KTD] := 0;
   	END_IF;
   END_IF;
   
   IF ETAPA8_D AND NOT ETAPA10_D THEN
   ETAPA8_D := 0;
   ETAPA9_D := 1;
   END_IF;
   
   IF ETAPA9_D THEN
   TCV_202_1 :=  VEC_U_D[KTD];  // Envio de valor de esfuerzo de control a la valvula de agua fria del intercambiador de calor 2
   END_IF;
   
   IF ETAPA9_D AND NOT ETAPA11_D THEN
   ETAPA9_D := 0;
   ETAPA10_D := 1;
   END_IF;
   
   IF ETAPA10_D THEN
   E2_D := E1_D;   // Actualizacion de errores pasados
   END_IF;
   
   IF ETAPA10_D AND NOT ETAPA12_D THEN
   ETAPA10_D := 0;
   ETAPA11_D := 1;
   END_IF;
   
   IF ETAPA11_D THEN
   E1_D := E0_D;    // Actualizacion de errores pasados
   END_IF;
   
   IF ETAPA11_D AND NOT ETAPA13_D THEN
   ETAPA11_D := 0;
   ETAPA12_D := 1;
   END_IF;
   
   IF ETAPA12_D THEN			// Desplazamiento de valores en el vector de la ley de control para actualizar valores pasados
   	FOR I_D:=1 TO KTD DO
   		VEC_U_D[I_D - 1] := VEC_U_D[I_D];
   	END_FOR;
   END_IF;
   
   IF ETAPA12_D AND NOT ETAPA14_D THEN
   ETAPA12_D := 0;
   ETAPA13_D := 1;
   END_IF;
   
   IF ETAPA13_D THEN
   Yn1_D := Yn_D;    // Actualizacion de valores pasados del modelo con retardo y el modelo rapido
   Yt1_D := Yt_D;
   END_IF;
   
   IF ETAPA13_D AND NOT ETAPA2_D THEN
   ETAPA13_D := 0;
   ETAPA14_D := 1;
   END_IF;
   
   IF ETAPA14_D THEN     // Tiempo de espera para recibir datos
   TONR(TIMER_DT);
   TIMER_DT.PRE := 2000;
   TIMER_DT.Reset := 0;
   TIMER_DT.TimerEnable := 1;
   END_IF;
   
END_ROUTINE
END_PROGRAM

PROGRAM Mapeo_CadSim_Plus   (* main routine Main *)

ROUTINE Main   (* ladder *)
END_ROUTINE

ROUTINE Mapeo1_DI   (* ladder *)
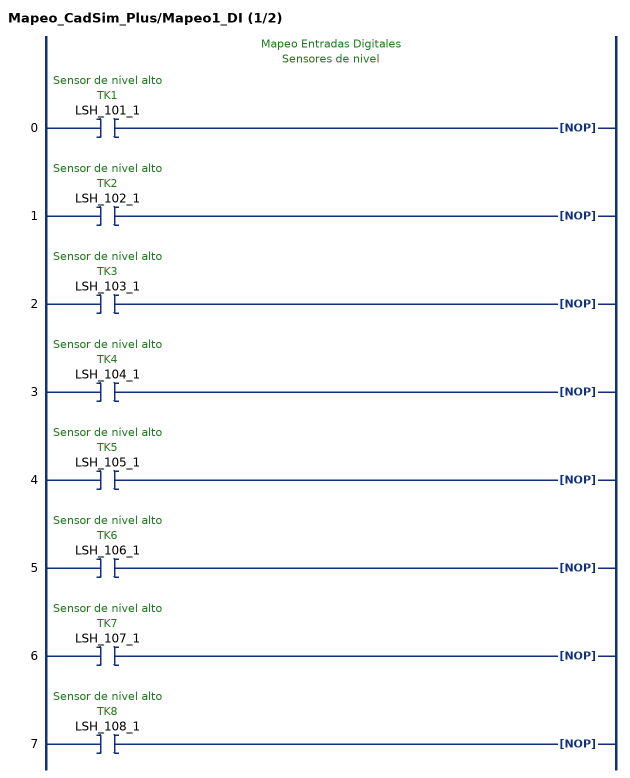
   // Mapeo Entradas Digitales
   // Sensores de nivel
   0: XIC(LSH_101_1)NOP();
   1: XIC(LSH_102_1)NOP();
   2: XIC(LSH_103_1)NOP();
   3: XIC(LSH_104_1)NOP();
   4: XIC(LSH_105_1)NOP();
   5: XIC(LSH_106_1)NOP();
   6: XIC(LSH_107_1)NOP();
   7: XIC(LSH_108_1)NOP();
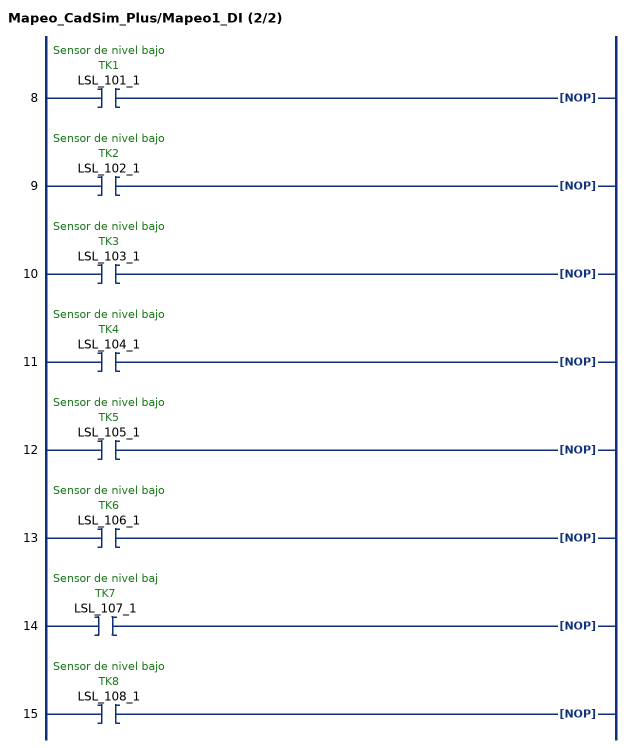
   8: XIC(LSL_101_1)NOP();
   9: XIC(LSL_102_1)NOP();
   10: XIC(LSL_103_1)NOP();
   11: XIC(LSL_104_1)NOP();
   12: XIC(LSL_105_1)NOP();
   13: XIC(LSL_106_1)NOP();
   14: XIC(LSL_107_1)NOP();
   15: XIC(LSL_108_1)NOP();
END_ROUTINE

ROUTINE Mapeo2_DO   (* ladder *)
END_ROUTINE

ROUTINE Mapeo3_AI   (* function block diagram *)
   SHEET 1
END_ROUTINE

ROUTINE Mapeo4_AO   (* ladder *)
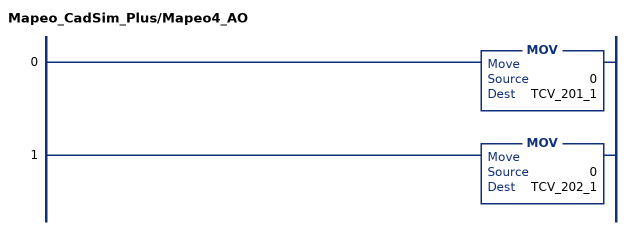
   0: MOV(0,TCV_201_1);
   1: MOV(0,TCV_202_1);
END_ROUTINE
END_PROGRAM
